(* CODESYS project Kruising Demo.project

Project tree, tasks and I/O mapping:
  Device : CODESYS Control Win V3, 3S - Smart Software Solutions GmbH, version 3.5.13.20
    application App
      libraries: Standard, 3.5.13.0 (System)
      task MainTask (cyclic, interval t#10ms, priority 1) calls Crossing_PRG
      program Crossing_PRG [ST]
      visualisation DeviceVisualization
      image pool CrossingImage
      global variables GVL
  libraries: VisuSymbols, 3.5.10.0 (System)
  interface ITrafficLight: goGreen, goRed, isRed
  interface ITrafficDetector: enable, isTriggered
  CrossingDevices/
    function block TrafficDetector [ST]: initialize, enable, isTriggered, cycle
    data type TrafficLightState
    GlobalImagePool
    function block TrafficLight [ST]: goGreen, goRed, isRed, initialize, cycle
    function block PedestrianLight [ST]: flashGreen
    data type DetectorState
  CrossingControl/
    function block Crossing [ST]: initialize, cycle
    data type LaneState
    function block Lane [ST]: cycle, someConflictsWaiting, initialize, allConflictsClosed, state
    interface ILane: State
  5ce3da45-db07-42e7-a21c-a00fff4ed8f6|F:\@@\Cursussen\OO-PLC programming\Lab\visu\crossing.gif
  5ce3da45-db07-42e7-a21c-a00fff4ed8f6|visu\crossing.gif
  text list GlobalTextList
*)

// CrossingControl/LaneState
TYPE LaneState :
(
	Closed, Waiting, Open, Closing
);
END_TYPE

// CrossingDevices/TrafficLightState
TYPE TrafficLightState :
(
	Red, Green, GreenExpired, Amber
);
END_TYPE

// CrossingDevices/DetectorState
TYPE DetectorState :
(
	Enabled, Disabled
);
END_TYPE

// Device/App/GVL
VAR_GLOBAL
	 CONSTANT iL : INT := 14;	  
	 aaConflictMatrix  : ARRAY [1..iL,1..iL] OF BOOL := 
[FALSE, FALSE, FALSE,  TRUE,  TRUE, FALSE, FALSE,  TRUE,  TRUE,  TRUE,   TRUE,  FALSE,  FALSE,  FALSE,
 FALSE, FALSE, FALSE,  TRUE,  TRUE,  TRUE,  TRUE, FALSE, FALSE,  TRUE,   TRUE,  FALSE,  FALSE,  FALSE,
 FALSE, FALSE, FALSE, FALSE, FALSE, FALSE,  TRUE, FALSE, FALSE, FALSE,   TRUE,  FALSE,   TRUE,   TRUE,
  TRUE,  TRUE, FALSE, FALSE, FALSE, FALSE,  TRUE,  TRUE, FALSE, FALSE,   TRUE,   TRUE,   TRUE,   TRUE, 
  TRUE,  TRUE, FALSE, FALSE, FALSE, FALSE,  TRUE,  TRUE,  TRUE,  TRUE,  FALSE,  FALSE,   TRUE,   TRUE,
 FALSE,  TRUE, FALSE, FALSE, FALSE, FALSE, FALSE, FALSE, FALSE,  TRUE,  FALSE,  FALSE,   TRUE,   TRUE,
 FALSE,  TRUE,  TRUE,  TRUE,  TRUE, FALSE, FALSE, FALSE, FALSE,  TRUE,   TRUE,  FALSE,   TRUE,   TRUE,
  TRUE, FALSE, FALSE,  TRUE,  TRUE, FALSE, FALSE, FALSE, FALSE,  TRUE,   TRUE,   TRUE,  FALSE,  FALSE,
  TRUE, FALSE, FALSE, FALSE,  TRUE, FALSE, FALSE, FALSE, FALSE, FALSE,  FALSE,  FALSE,  FALSE,  FALSE,
  TRUE,  TRUE, FALSE, FALSE,  TRUE,  TRUE,  TRUE,  TRUE, FALSE, FALSE,  FALSE,  FALSE,  FALSE,  FALSE,
  TRUE,  TRUE,  TRUE,  TRUE, FALSE, FALSE,  TRUE,  TRUE, FALSE, FALSE,  FALSE,  FALSE,   TRUE,   TRUE,
 FALSE, FALSE, FALSE,  TRUE, FALSE, FALSE, FALSE,  TRUE, FALSE, FALSE,  FALSE,  FALSE,  FALSE,  FALSE,
 FALSE, FALSE,  TRUE,  TRUE,  TRUE,  TRUE,  TRUE, FALSE, FALSE, FALSE,   TRUE,  FALSE,  FALSE,  FALSE,
 FALSE, FALSE,  TRUE,  TRUE,  TRUE,  TRUE,  TRUE, FALSE, FALSE, FALSE,   TRUE,  FALSE,  FALSE,  FALSE];
END_VAR

// Device/App/Crossing_PRG
PROGRAM Crossing_PRG
VAR
	oCrossing: Crossing;
	xInitialized : BOOL := FALSE;
END_VAR

//Initialize aggregated objects
IF NOT xInitialized THEN
 	oCrossing.initialize();
	xInitialized := TRUE;
END_IF

// Activate active objects
oCrossing.cycle();

END_PROGRAM

// CrossingControl/Crossing
FUNCTION_BLOCK Crossing
VAR
	aoDetector : ARRAY [1..14] OF TrafficDetector;
    aoLight : ARRAY [1..12] OF TrafficLight;
	oLight13 : PedestrianLight;
	oLight14 : PedestrianLight;
	aoLane : ARRAY [1..14] OF Lane;	
END_VAR

METHOD initialize
VAR	
	iJ: INT;
	apLane : ARRAY [1..14] OF ILane;	
END_VAR
// Initialize aggregated objects
FOR iJ:= 1 TO 14 DO
	aoDetector[iJ].initialize();
END_FOR;
FOR iJ:= 1 TO 12 DO
	aoLight[iJ].initialize();
END_FOR;
oLight13.initialize();
oLight14.initialize();
FOR iJ:= 1 TO 14 DO
	apLane[iJ] := aoLane[iJ];
END_FOR;
FOR iJ:= 1 TO 12 DO
	aolane[iJ].initialize(iJ, aoDetector[iJ], aoLight[iJ], apLane);
END_FOR;
aoLane[13].initialize(13, aoDetector[13], oLight13, apLane);
aoLane[14].initialize(14, aoDetector[14], oLight14, apLane);
END_METHOD

METHOD cycle
VAR
	iJ: INT;
END_VAR
// cycle through aggregated objects

FOR iJ:= 1 TO 12 DO
	aoLight[iJ].cycle();
END_FOR;
oLight13.cycle();
oLight14.cycle();
FOR iJ:= 1 TO 14 DO
	aoDetector[iJ].cycle();
	aolane[iJ].cycle();
END_FOR;
END_METHOD

END_FUNCTION_BLOCK

// CrossingDevices/TrafficDetector
FUNCTION_BLOCK TrafficDetector IMPLEMENTS ITrafficDetector
VAR
	xTriggered : BOOL := FALSE;
	eState: DetectorState;
END_VAR

// Cycle through aggregated objects
 	// There are none

// Transitions for this state machine

IF xTriggered THEN
	eState := Disabled;
END_IF

METHOD PUBLIC initialize
// Initialize attribute values
xTriggered:=FALSE;
eState := Enabled;

//No aggregated objects
END_METHOD

METHOD PUBLIC enable
IF xTriggered THEN
	xTriggered := FALSE;
	eState := Enabled;
END_IF
END_METHOD

METHOD PUBLIC isTriggered : BOOL
isTriggered := xTriggered;
END_METHOD

METHOD cycle
THIS^();
END_METHOD

END_FUNCTION_BLOCK

// ITrafficDetector
INTERFACE ITrafficDetector

METHOD enable
END_METHOD

METHOD isTriggered : BOOL
END_METHOD

END_INTERFACE

// CrossingDevices/TrafficLight
FUNCTION_BLOCK TrafficLight IMPLEMENTS ITrafficLight
VAR
	xRedOn : BOOL;
	xGreenOn : BOOL;
	xAmberOn : BOOL;
	xRedRequested : BOOL;
	tGreenTimer : TON;
	tAmberTimer : TON;
	eState : TrafficLightState;	
END_VAR

// cycle through aggregated objects
tGreenTimer(IN:=(eState=Green),PT:=T#10S);
tAmberTimer(IN:=(eState=Amber),PT:=T#5S);

// transitions for this state machine

CASE eState OF
Red: // call event handled in goGreen()
Green:
	IF tGreenTimer.Q THEN
		eState := GreenExpired;
	END_IF
GreenExpired: // call event handled in goRed()		
	IF xRedRequested THEN
		xGreenOn := FALSE;				
		xRedRequested := FALSE;		
		eState := Amber;
		xAmberOn := TRUE;
	END_IF
Amber:
	IF tAmberTimer.Q THEN
		xAmberOn := FALSE;
		eState := Red;
		xRedOn := TRUE;		
	END_IF
END_CASE

METHOD PUBLIC goGreen
CASE eState OF
Red:
	xRedOn := FALSE;
	eState := Green;
	xGreenOn := TRUE;	
END_CASE
END_METHOD

METHOD PUBLIC goRed
CASE eState OF
Green:
	xRedRequested := TRUE;
GreenExpired:
	xGreenOn := FALSE;
	eState := Amber;
	xAmberOn := TRUE;	
END_CASE
END_METHOD

METHOD PUBLIC isRed : BOOL
isRed := xRedOn;
END_METHOD

METHOD PUBLIC initialize
// initialize attributes
eState := Red;
xRedOn := TRUE;

// initialize aggregated objects
   // No aggregated objects
END_METHOD

METHOD cycle
THIS^();
END_METHOD

END_FUNCTION_BLOCK

// ITrafficLight
INTERFACE ITrafficLight

METHOD  goGreen
END_METHOD

METHOD goRed
END_METHOD

METHOD isRed : BOOL
END_METHOD

END_INTERFACE

// CrossingDevices/PedestrianLight
FUNCTION_BLOCK PedestrianLight EXTENDS TrafficLight
VAR
	tOffTimer : TON;
	tOnTimer : TON;
END_VAR

// cycle through aggregated objects
tOnTimer(IN:=(eState=Amber AND xGreenOn),PT:=T#1S);
tOffTimer(IN:=(eState=Amber AND NOT xGreenOn),PT:=T#1S);

// cycle through the parent
SUPER^();

// transitions for this state machine

CASE eState OF
Amber:
	flashGreen();
END_CASE

METHOD PRIVATE flashGreen
IF tOnTimer.Q THEN
	xGreenOn := FALSE;
END_IF
IF tOffTimer.Q THEN
	xGreenOn := TRUE;
END_IF
END_METHOD

END_FUNCTION_BLOCK

// CrossingControl/Lane
FUNCTION_BLOCK Lane IMPLEMENTS ILane
VAR
	iN : INT;
    eState : LaneState;		
	pLight : ITrafficLight;
	pDetector : ITrafficDetector;
    apPeer : ARRAY [1..GVL.iL] OF ILane;
END_VAR

// Perform transitions for this state machine 

CASE eState OF 
Closed: 
 	IF pDetector.isTriggered()  THEN
		eState := Waiting;
	END_IF
Waiting : 
	IF allConflictsClosed() THEN
		eState := Open;
		pLight.goGreen();		
	END_IF
Open :
	IF someConflictsWaiting() THEN
		eState := Closing;
		pLight.goRed();		
	END_IF 
Closing :
	IF pLight.isRed() THEN 
		eState := Closed;
		pDetector.enable();		
	END_IF 
END_CASE

METHOD PUBLIC cycle
THIS^();

// Activate aggregated objects
    // only interfaces
END_METHOD

METHOD PRIVATE someConflictsWaiting : BOOL
VAR
	iJ: INT;
END_VAR
someConflictsWaiting := TRUE;
FOR iJ:=1 TO GVL.iL DO
	IF aaConflictMatrix[iJ,iN] THEN
		IF apPeer[iJ].state = Waiting THEN
			RETURN;
		END_IF
	END_IF
END_FOR;
someConflictsWaiting := FALSE;
END_METHOD

METHOD PUBLIC initialize
VAR_INPUT
	iJ : INT;
	pD : ITrafficDetector;
	pL : ITrafficLight; 
	apIn : ARRAY [1..14] OF ILane;
END_VAR
// Initialize attribute values
iN:=iJ;
eState := Closed;
pLight := pL;
pDetector := pD;
apPeer := apIn;

// Initialize aggregated objects
END_METHOD

METHOD PRIVATE allConflictsClosed : BOOL
VAR
	iJ: INT;
END_VAR
allConflictsClosed := FALSE;
FOR iJ:=1 TO GVL.iL DO
	IF aaConflictMatrix[iJ,iN] THEN
		IF apPeer[iJ].state = Open OR apPeer[iJ].state=Closing THEN
			RETURN;
		END_IF
	END_IF
END_FOR;
allConflictsClosed:= TRUE;
END_METHOD

PROPERTY PUBLIC state : LaneState
GET
state := eState;
END_GET
END_PROPERTY

END_FUNCTION_BLOCK

// CrossingControl/ILane
INTERFACE ILane

PROPERTY State : LaneState
GET
END_GET
END_PROPERTY

END_INTERFACE

// Device/App/DeviceVisualization
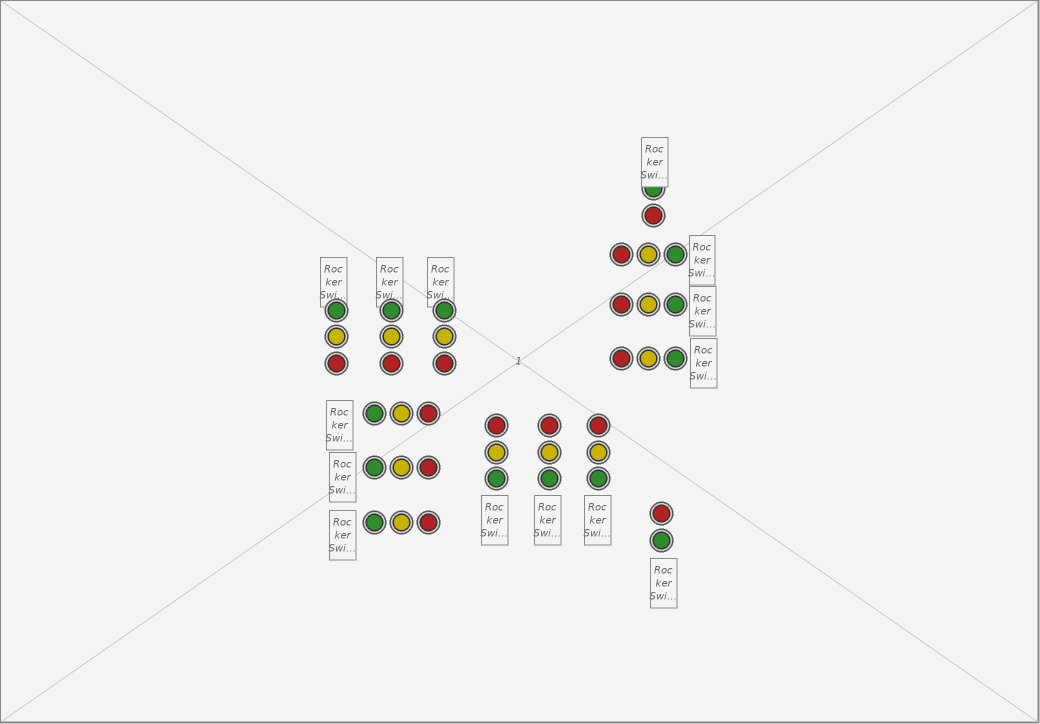
VISUALIZATION DeviceVisualization  // 1040x724, background image 0
    Image (0,0 1038x722), image: 1
    Lamp1 (648,527 27x27), variable: Crossing_PRG.oCrossing.oLight13.xGreenOn, style: Lamp-Lamp1-Green
    Lamp1 (648,500 27x27), variable: Crossing_PRG.oCrossing.oLight13.xRedOn, style: Lamp-Lamp1-Red
    Lamp1 (640,175 27x27), variable: Crossing_PRG.oCrossing.oLight14.xGreenOn, style: Lamp-Lamp1-Green
    Lamp1 (640,202 27x27), variable: Crossing_PRG.oCrossing.oLight14.xRedOn, style: Lamp-Lamp1-Red
    RockerSwitch (481,495 27x50), variable: Crossing_PRG.oCrossing.aoDetector[1].xTriggered, input disabled if: Crossing_PRG.oCrossing.aoDetector[1].xTriggered, behaviour: TOGGLE, style: Switch-RockerSwitch-Gray
    RockerSwitch (534,495 27x50), variable: Crossing_PRG.oCrossing.aoDetector[2].xTriggered, input disabled if: Crossing_PRG.oCrossing.aoDetector[2].xTriggered, behaviour: TOGGLE, style: Switch-RockerSwitch-Gray
    RockerSwitch (584,495 27x50), variable: Crossing_PRG.oCrossing.aoDetector[3].xTriggered, input disabled if: Crossing_PRG.oCrossing.aoDetector[3].xTriggered, behaviour: TOGGLE, style: Switch-RockerSwitch-Gray
    RockerSwitch (690,338 27x50), variable: Crossing_PRG.oCrossing.aoDetector[4].xTriggered, input disabled if: Crossing_PRG.oCrossing.aoDetector[4].xTriggered, behaviour: TOGGLE, style: Switch-RockerSwitch-Gray
    RockerSwitch (689,286 27x50), variable: Crossing_PRG.oCrossing.aoDetector[5].xTriggered, input disabled if: Crossing_PRG.oCrossing.aoDetector[5].xTriggered, behaviour: TOGGLE, style: Switch-RockerSwitch-Gray
    RockerSwitch (689,235 26x50), variable: Crossing_PRG.oCrossing.aoDetector[6].xTriggered, input disabled if: Crossing_PRG.oCrossing.aoDetector[6].xTriggered, behaviour: TOGGLE, style: Switch-RockerSwitch-Gray
    RockerSwitch (427,257 27x50), variable: Crossing_PRG.oCrossing.aoDetector[7].xTriggered, input disabled if: Crossing_PRG.oCrossing.aoDetector[7].xTriggered, behaviour: TOGGLE, style: Switch-RockerSwitch-Gray
    RockerSwitch (376,257 27x50), variable: Crossing_PRG.oCrossing.aoDetector[8].xTriggered, input disabled if: Crossing_PRG.oCrossing.aoDetector[8].xTriggered, behaviour: TOGGLE, style: Switch-RockerSwitch-Gray
    RockerSwitch (320,257 27x50), variable: Crossing_PRG.oCrossing.aoDetector[9].xTriggered, input disabled if: Crossing_PRG.oCrossing.aoDetector[9].xTriggered, behaviour: TOGGLE, style: Switch-RockerSwitch-Gray
    RockerSwitch (326,400 27x50), variable: Crossing_PRG.oCrossing.aoDetector[10].xTriggered, input disabled if: Crossing_PRG.oCrossing.aoDetector[10].xTriggered, behaviour: TOGGLE, style: Switch-RockerSwitch-Gray
    RockerSwitch (329,452 27x50), variable: Crossing_PRG.oCrossing.aoDetector[11].xTriggered, input disabled if: Crossing_PRG.oCrossing.aoDetector[11].xTriggered, behaviour: TOGGLE, style: Switch-RockerSwitch-Gray
    RockerSwitch (329,510 27x50), variable: Crossing_PRG.oCrossing.aoDetector[12].xTriggered, input disabled if: Crossing_PRG.oCrossing.aoDetector[12].xTriggered, behaviour: TOGGLE, style: Switch-RockerSwitch-Gray
    RockerSwitch (650,558 27x50), variable: Crossing_PRG.oCrossing.aoDetector[13].xTriggered, input disabled if: Crossing_PRG.oCrossing.aoDetector[13].xTriggered, behaviour: TOGGLE, style: Switch-RockerSwitch-Gray
    RockerSwitch (641,137 27x50), variable: Crossing_PRG.oCrossing.aoDetector[14].xTriggered, input disabled if: Crossing_PRG.oCrossing.aoDetector[14].xTriggered, behaviour: TOGGLE, style: Switch-RockerSwitch-Gray
    Lamp1 (483,439 27x27), variable: Crossing_PRG.oCrossing.aoLight[1].xAmberOn, style: Lamp-Lamp1-Yellow
    Lamp1 (483,465 27x27), variable: Crossing_PRG.oCrossing.aoLight[1].xGreenOn, style: Lamp-Lamp1-Green
    Lamp1 (483,412 27x27), variable: Crossing_PRG.oCrossing.aoLight[1].xRedOn, style: Lamp-Lamp1-Red
    Lamp1 (536,439 27x27), variable: Crossing_PRG.oCrossing.aoLight[2].xAmberOn, style: Lamp-Lamp1-Yellow
    Lamp1 (536,465 27x27), variable: Crossing_PRG.oCrossing.aoLight[2].xGreenOn, style: Lamp-Lamp1-Green
    Lamp1 (536,412 27x27), variable: Crossing_PRG.oCrossing.aoLight[2].xRedOn, style: Lamp-Lamp1-Red
    Lamp1 (585,439 27x27), variable: Crossing_PRG.oCrossing.aoLight[3].xAmberOn, style: Lamp-Lamp1-Yellow
    Lamp1 (585,465 27x27), variable: Crossing_PRG.oCrossing.aoLight[3].xGreenOn, style: Lamp-Lamp1-Green
    Lamp1 (585,412 27x27), variable: Crossing_PRG.oCrossing.aoLight[3].xRedOn, style: Lamp-Lamp1-Red
    Lamp1 (431,323 27x27), variable: Crossing_PRG.oCrossing.aoLight[7].xAmberOn, style: Lamp-Lamp1-Yellow
    Lamp1 (431,297 27x27), variable: Crossing_PRG.oCrossing.aoLight[7].xGreenOn, style: Lamp-Lamp1-Green
    Lamp1 (431,350 27x27), variable: Crossing_PRG.oCrossing.aoLight[7].xRedOn, style: Lamp-Lamp1-Red
    Lamp1 (378,323 27x27), variable: Crossing_PRG.oCrossing.aoLight[8].xAmberOn, style: Lamp-Lamp1-Yellow
    Lamp1 (378,297 27x27), variable: Crossing_PRG.oCrossing.aoLight[8].xGreenOn, style: Lamp-Lamp1-Green
    Lamp1 (378,350 27x27), variable: Crossing_PRG.oCrossing.aoLight[8].xRedOn, style: Lamp-Lamp1-Red
    Lamp1 (323,323 27x27), variable: Crossing_PRG.oCrossing.aoLight[9].xAmberOn, style: Lamp-Lamp1-Yellow
    Lamp1 (323,297 27x27), variable: Crossing_PRG.oCrossing.aoLight[9].xGreenOn, style: Lamp-Lamp1-Green
    Lamp1 (323,350 27x27), variable: Crossing_PRG.oCrossing.aoLight[9].xRedOn, style: Lamp-Lamp1-Red
    Lamp1 (635,291 27x27), variable: Crossing_PRG.oCrossing.aoLight[5].xAmberOn, style: Lamp-Lamp1-Yellow
    Lamp1 (662,291 27x27), variable: Crossing_PRG.oCrossing.aoLight[5].xGreenOn, style: Lamp-Lamp1-Green
    Lamp1 (608,291 27x27), variable: Crossing_PRG.oCrossing.aoLight[5].xRedOn, style: Lamp-Lamp1-Red
    Lamp1 (635,241 27x27), variable: Crossing_PRG.oCrossing.aoLight[6].xAmberOn, style: Lamp-Lamp1-Yellow
    Lamp1 (662,241 27x27), variable: Crossing_PRG.oCrossing.aoLight[6].xGreenOn, style: Lamp-Lamp1-Green
    Lamp1 (608,241 27x27), variable: Crossing_PRG.oCrossing.aoLight[6].xRedOn, style: Lamp-Lamp1-Red
    Lamp1 (635,345 27x27), variable: Crossing_PRG.oCrossing.aoLight[4].xAmberOn, style: Lamp-Lamp1-Yellow
    Lamp1 (662,345 27x27), variable: Crossing_PRG.oCrossing.aoLight[4].xGreenOn, style: Lamp-Lamp1-Green
    Lamp1 (608,345 27x27), variable: Crossing_PRG.oCrossing.aoLight[4].xRedOn, style: Lamp-Lamp1-Red
    Lamp1 (388,509 27x27), variable: Crossing_PRG.oCrossing.aoLight[12].xAmberOn, style: Lamp-Lamp1-Yellow
    Lamp1 (361,509 27x27), variable: Crossing_PRG.oCrossing.aoLight[12].xGreenOn, style: Lamp-Lamp1-Green
    Lamp1 (415,509 27x27), variable: Crossing_PRG.oCrossing.aoLight[12].xRedOn, style: Lamp-Lamp1-Red
    Lamp1 (388,454 27x27), variable: Crossing_PRG.oCrossing.aoLight[11].xAmberOn, style: Lamp-Lamp1-Yellow
    Lamp1 (361,454 27x27), variable: Crossing_PRG.oCrossing.aoLight[11].xGreenOn, style: Lamp-Lamp1-Green
    Lamp1 (415,454 27x27), variable: Crossing_PRG.oCrossing.aoLight[11].xRedOn, style: Lamp-Lamp1-Red
    Lamp1 (388,400 27x27), variable: Crossing_PRG.oCrossing.aoLight[10].xAmberOn, style: Lamp-Lamp1-Yellow
    Lamp1 (361,400 27x27), variable: Crossing_PRG.oCrossing.aoLight[10].xGreenOn, style: Lamp-Lamp1-Green
    Lamp1 (415,400 27x27), variable: Crossing_PRG.oCrossing.aoLight[10].xRedOn, style: Lamp-Lamp1-Red
END_VISUALIZATION
